FUNCTION_BLOCK StepRestOfTimeCalc2 (* Basic Function Block Type *)
  (* Standard: 61499-2 *)
  (* Version 0.0, 7/15/2026, Schneider Electric, Template *)
  PACKAGE SE.Nereda;
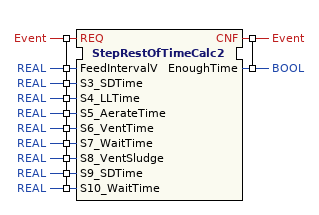
  EVENT_INPUT
    REQ WITH FeedIntervalV, S3_SDTime, S4_LLTime, S5_AerateTime, S6_VentTime, S7_WaitTime, S8_VentSludge, S9_SDTime, S10_WaitTime; (* Normal Execution Request *)
  END_EVENT
  EVENT_OUTPUT
    CNF WITH EnoughTime; (* Execution Confirmation *)
  END_EVENT
  VAR_INPUT
    FeedIntervalV : REAL;
    S3_SDTime : REAL;
    S4_LLTime : REAL;
    S5_AerateTime : REAL;
    S6_VentTime : REAL;
    S7_WaitTime : REAL;
    S8_VentSludge : REAL;
    S9_SDTime : REAL;
    S10_WaitTime : REAL;
  END_VAR
  VAR_OUTPUT
    EnoughTime : BOOL;
  END_VAR
  VAR
    RestOfTime : REAL;
    SDTime : REAL;
  END_VAR
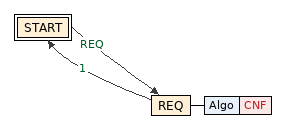
  EC_STATES
    START; (* Initial State *)
    REQ : Algo -> CNF; (* Normal execution *)
  END_STATES
  EC_TRANSITIONS
    START TO REQ := REQ;
    REQ TO START := 1;
  END_TRANSITIONS
  ALGORITHM Algo IN ST:
;
IF S3_SDTime >= S9_SDTime THEN
	SDTime := S3_SDTime;
ELSE
	SDTime := S9_SDTime;
END_IF;

RestOfTime := FeedIntervalV - (SDTime + S4_LLTime + S5_AerateTime + S6_VentTime + S7_WaitTime + S8_VentSludge + S10_WaitTime);

IF RestOfTime < 0 THEN
	EnoughTime := FALSE;
ELSE
	EnoughTime := TRUE;
END_IF;
  END_ALGORITHM
END_FUNCTION_BLOCK
